TYPE E_SafetyState :
(
	Idle,
	RestoreReference,
	VerifyReference,
	Homing,
	MoveToZero,
	Complete,
	ProtectiveStop,
	ErrorStop
);
END_TYPE

(* stored: Version 1.1.0.1, ProductVersion 3.1.4024.15
   DUT E_SafetyState: Id {21615fb9-b894-4865-bfdc-591d3f979594} *)
